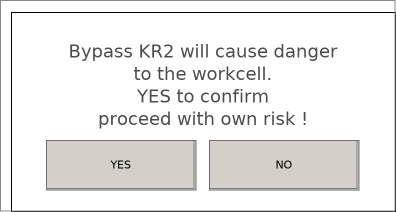
VISUALIZATION MSG_KR2_BP  // 396x212
    RoundedRectangle (11,12 385x200)
    Button (46,140 150x50), "YES"
        OnMouseClick: CloseDialog Dialog=MSG_KR2_BP, Result=Yes, NumpadKeypadSet=True
        OnMouseClick: execute { GVL.KR2_bypass := TRUE; }
    Button (209,140 150x50), "NO"
        OnMouseClick: execute { GVL.KR2_bypass := FALSE; }
        OnMouseClick: CloseDialog Dialog=MSG_KR2_BP, Result=No, NumpadKeypadSet=True
    Label (55,30 296x110), "Bypass KR2 will cause danger to the workcell. YES to confirm proceed with own risk !"
END_VISUALIZATION

(* stored: Version 1.1.0.1, ProductVersion 3.1.4024.12
   Visu MSG_KR2_BP: Id {0aa862f5-5d2a-4774-8059-4491ea4d6a44} *)
